{attribute addProperty BoxType "EK1100-0000-0018"}
{attribute addProperty Id "Beckhoff_EPP2xxxEK1122Beckhoff_EPP2xxxEK1122_A6F06543168002100"}
{attribute addProperty CRC "3066888283"}
{attribute addProperty SizeInBites "16800"}
{attribute addProperty SizeInBytes "2100"}
TYPE Beckhoff_EPP2xxx_B6CD005B EXTENDS EK1100_179A0949 :
STRUCT
	{attribute addProperty Name "Beckhoff_EPP2xxxEK1122"}
	Beckhoff_EPP2xxxEK1122 : Beckhoff_EPP2xxxEK1122_A6F06543;
END_STRUCT
END_TYPE

(* stored: Version 1.2.0.0, ProductVersion 3.1.4024.9
   DUT Beckhoff_EPP2xxx_B6CD005B: Id {1e9787ac-0ae4-4d9c-acfa-f1017d0cc328} *)
